FUNCTION_BLOCK Pump EXTENDS Motor
VAR_INPUT
END_VAR
VAR_OUTPUT
END_VAR
VAR
END_VAR

iPapaTime(in:=xOn, pt:=T#1S);
UpdateAngle();

METHOD UpdateAngle : BOOL
VAR_INPUT
END_VAR
IF ipapatime.q THEN
	//iangle:= iangle+ispeed;
	iangle:= iangle+ispeed*100;
//	IF iangle>360 THEN
//		iangle:=0;
//	END_IF
	ipapatime.IN:= FALSE;
ELSE
	ipapatime.IN:= TRUE;
END_IF
END_METHOD

END_FUNCTION_BLOCK

(* stored: Version 1.1.0.1, ProductVersion 3.1.4024.12
   POU Pump: Id {86477610-007c-4c65-b262-d72fd6793daa}, SpecialFunc None
   Method UpdateAngle: Id {debe4aeb-b848-49f8-82a3-2e88c667bf22} *)
